(* CODESYS project tc3_hbi_cylinder.library
   Placeholder: Tc3_HBI_Cylinder
   Title: Tc3_HBI_Cylinder
   Version: 3.5.3.6
   DefaultNamespace: Tc3_HBI_Cylinder
   Company: BeckHoff SG

Project tree, tasks and I/O mapping:
  libraries: Tc2_Standard, * (Beckhoff Automation GmbH); Tc2_System, * (Beckhoff Automation GmbH); Tc2_Utilities, * (Beckhoff Automation GmbH); Tc3_HBI_System, * (BeckHoff)
  04_Cylinder/
    DUTs/
      data type _ST_Cylinder
      data type _ST_Cylinder_Status
      data type ST_Cylinder
    ITFs/
      interface I_Cylinder: M_nExtend, M_nOff, M_nRetract, M_nSetOutputOff, P_ipExtend, P_ipRetract, P_nExtendAlarmID, P_nRetractAlarmID, P_opExtend, P_opRetract, P_SensorDelay, P_sExtAlarmDesc, P_sMessage, P_sRetAlarmDesc, P_Timeout
    POUs/
      function block FB_Cylinder [ST]: M_nExtend, M_nOff, M_nReset, M_nRetract, M_nSetOutputOff, P_ipExtend, P_ipRetract, P_nExtendAlarmID, P_nRetractAlarmID, P_opExtend, P_opRetract, P_SensorDelay, P_sExtAlarmDesc, P_sMessage, P_sRetAlarmDesc, P_Timeout
  05_Vacuum/
    DUTs/
      data type _ST_Vacuum
      data type _ST_Vacuum_Status
      data type ST_Vacuum
    ITFs/
      interface I_Vacuum: M_nOff, M_nSetOutputOff, M_nVacuumOff, M_nVacuumOn, P_ipVacuumOff, P_ipVacuumOn, P_nVacOffAlarmID, P_nVacOnAlarmID, P_opVacuumOff, P_opVacuumOn, P_SensorDelay, P_sMessage, P_sVacOffAlarmDesc, P_sVacOnAlarmDesc, P_Timeout
    POUs/
      function block FB_Vacuum [ST]: M_nOff, M_nReset, M_nSetOutputOff, M_nVacuumOff, M_nVacuumOn, P_ipVacuumOff, P_ipVacuumOn, P_nVacOffAlarmID, P_nVacOnAlarmID, P_opVacuumOff, P_opVacuumOn, P_SensorDelay, P_sMessage, P_sVacOffAlarmDesc, P_sVacOnAlarmDesc, P_Timeout
  06_Purge/
    DUTs/
      data type _ST_Purge
      data type _ST_Purge_Status
      data type ST_Purge
    ITFs/
      interface I_Purge: M_nOff, M_nPurgeOff, M_nPurgeOn, M_nSetOutputOff, P_ipPurgeOff, P_ipPurgeOn, P_nPurgeOffAlarmID, P_nPurgeOnAlarmID, P_opPurgeOff, P_opPurgeOn, P_SensorDelay, P_sMessage, P_sPurgeOffAlarmDesc, P_sPurgeOnAlarmDesc, P_Timeout
    POUs/
      function block FB_Purge [ST]: M_nOff, M_nPurgeOff, M_nPurgeOn, M_nReset, M_nSetOutputOff, P_ipPurgeOff, P_ipPurgeOn, P_nPurgeOffAlarmID, P_nPurgeOnAlarmID, P_opPurgeOff, P_opPurgeOn, P_SensorDelay, P_sMessage, P_sPurgeOffAlarmDesc, P_sPurgeOnAlarmDesc, P_Timeout
  07_VacuumPurge/
    DUTs/
      data type _ST_VacuumPurge
      data type _ST_VacuumPurge_Status
      data type ST_VacuumPurge
    ITFs/
      interface I_VacuumPurge: M_nNeutral, M_nPurgeOn, M_nVacuumOn
    POUs/
      function block FB_VacuumPurge [ST]: M_nNeutral, M_nOff, M_nPurgeOff, M_nPurgeOn, M_nSetOutputOff, M_nVacuumOff, M_nVacuumOn, P_ipPurgeOff, P_ipPurgeOn, P_ipVacuumOff, P_ipVacuumOn, P_nPurgeOffAlarmID, P_nPurgeOnAlarmID, P_nVacOffAlarmID, P_nVacOnAlarmID, P_opPurgeOff, P_opPurgeOn, P_opVacuumOff, P_opVacuumOn, P_PurgeTimeout, P_SensorDelay, P_sMessage, P_sPurgeOffAlarmDesc, P_sPurgeOnAlarmDesc, P_sVacOffAlarmDesc, P_sVacOnAlarmDesc, P_Timeout, P_VacuumTimeout
  Version/
    global variables Global_Version
*)

// 04_Cylinder/DUTs/_ST_Cylinder
TYPE _ST_Cylinder EXTENDS ST_Basic :
STRUCT
	;
END_STRUCT
END_TYPE

// 04_Cylinder/DUTs/_ST_Cylinder_Status
TYPE _ST_Cylinder_Status :
STRUCT
	ipExtend	: BOOL;
	ipRetract	: BOOL;
	opExtend	: BOOL;
	opRetract	: BOOL;
	M_nExtend: UDINT;
	M_nRetract: UDINT;
	M_nOff: UDINT;
END_STRUCT
END_TYPE

// 04_Cylinder/DUTs/ST_Cylinder
TYPE ST_Cylinder EXTENDS ST_Basic :
STRUCT
	bExtend		: BOOL;
	bRetract	: BOOL;
	udiExtendAlarmID: UDINT;
	udiRetractAlarmID: UDINT;
	sExtendAlarmDesc: STRING(80);
	sRetractAlarmDesc: STRING(80);
	sMessage: STRING(80);
	Timeout	: TIME:= T#5S;
	SensorDelay: TIME:= T#3S;
	stStatus: _ST_Cylinder_Status;
END_STRUCT
END_TYPE

// 05_Vacuum/DUTs/_ST_Vacuum
TYPE _ST_Vacuum EXTENDS ST_Basic :
STRUCT
	;
END_STRUCT
END_TYPE

// 05_Vacuum/DUTs/_ST_Vacuum_Status
TYPE _ST_Vacuum_Status :
STRUCT
	ipVacuumOn		: BOOL;
	ipVacuumOff		: BOOL;
	opVacuumOn		: BOOL;
	opVacuumOff		: BOOL;
	M_nVacuumOff: UDINT;
	M_nVacuumOn: UDINT;
	M_nOff: UDINT;
END_STRUCT
END_TYPE

// 05_Vacuum/DUTs/ST_Vacuum
TYPE ST_Vacuum EXTENDS ST_Basic :
STRUCT
	bVacuumOn		: BOOL;
	bVacuumOff		: BOOL;
	udiVacOffAlarmID: UDINT;
	udiVacOnAlarmID: UDINT;
	sVacOffAlarmDesc: STRING(80);
	sVacOnAlarmDesc: STRING(80);
	sMessage: STRING(80);
	Timeout	: TIME:= T#5S;
	SensorDelay: TIME:= T#3S;
	stStatus: _ST_Vacuum_Status;
END_STRUCT
END_TYPE

// 06_Purge/DUTs/_ST_Purge
TYPE _ST_Purge EXTENDS ST_Basic :
STRUCT
	;
END_STRUCT
END_TYPE

// 06_Purge/DUTs/_ST_Purge_Status
TYPE _ST_Purge_Status :
STRUCT
	ipPurgeOn		: BOOL;
	ipPurgeOff		: BOOL;
	opPurgeOn		: BOOL;
	opPurgeOff		: BOOL;
	M_nPurgeOff: UDINT;
	M_nPurgeOn: UDINT;
	M_nOff: UDINT;
END_STRUCT
END_TYPE

// 06_Purge/DUTs/ST_Purge
TYPE ST_Purge EXTENDS ST_Basic :
STRUCT
	bPurgeOn		: BOOL;
	bPurgeOff		: BOOL;
	udiPurgeOffAlarmID: UDINT;
	udiPurgeOnAlarmID: UDINT;
	sPurgeOffAlarmDesc: STRING(80);
	sPurgeOnAlarmDesc: STRING(80);
	sMessage: STRING(80);
	Timeout		: TIME:= T#5S;
	SensorDelay	: TIME:= T#3S;	
	stStatus: _ST_Purge_Status;
END_STRUCT
END_TYPE

// 07_VacuumPurge/DUTs/_ST_VacuumPurge
TYPE _ST_VacuumPurge EXTENDS _ST_Purge :
STRUCT
	;
END_STRUCT
END_TYPE

// 07_VacuumPurge/DUTs/_ST_VacuumPurge_Status
TYPE _ST_VacuumPurge_Status :
STRUCT
	;
END_STRUCT
END_TYPE

// 07_VacuumPurge/DUTs/ST_VacuumPurge
TYPE ST_VacuumPurge :
STRUCT
	;
END_STRUCT
END_TYPE

// Version/Global_Version
{attribute 'TcGenerated'}
{attribute 'no-analysis'}
{attribute 'linkalways'}
// This function has been automatically generated from the project information.
VAR_GLOBAL CONSTANT
	{attribute 'const_non_replaced'}
	stLibVersion_Tc3_HBI_Cylinder : ST_LibVersion := (iMajor := 3, iMinor := 5, iBuild := 3, iRevision := 6, sVersion := '3.5.3.6');
END_VAR

// 04_Cylinder/ITFs/I_Cylinder
INTERFACE I_Cylinder EXTENDS Tc3_HBI_System.I_Basic

METHOD M_nExtend : UDINT
VAR_INPUT
	bExecute: BOOL;
END_VAR
END_METHOD

METHOD M_nOff : UDINT
VAR_INPUT
END_VAR
END_METHOD

METHOD M_nRetract : UDINT
VAR_INPUT
	bExecute: BOOL;
END_VAR
END_METHOD

METHOD M_nSetOutputOff : UDINT
VAR_INPUT
END_VAR
END_METHOD

PROPERTY P_ipExtend : BOOL
GET
END_GET
SET
END_SET
END_PROPERTY

PROPERTY P_ipRetract : BOOL
GET
END_GET
SET
END_SET
END_PROPERTY

PROPERTY P_nExtendAlarmID : UDINT
SET
END_SET
END_PROPERTY

PROPERTY P_nRetractAlarmID : UDINT
SET
END_SET
END_PROPERTY

PROPERTY P_opExtend : BOOL
GET
END_GET
SET
END_SET
END_PROPERTY

PROPERTY P_opRetract : BOOL
GET
END_GET
SET
END_SET
END_PROPERTY

PROPERTY P_SensorDelay : TIME
SET
END_SET
END_PROPERTY

PROPERTY P_sExtAlarmDesc : STRING
SET
END_SET
END_PROPERTY

PROPERTY P_sMessage : STRING
GET
END_GET
END_PROPERTY

PROPERTY P_sRetAlarmDesc : STRING
SET
END_SET
END_PROPERTY

PROPERTY P_Timeout : TIME
SET
END_SET
END_PROPERTY

END_INTERFACE

// 04_Cylinder/POUs/FB_Cylinder
//------------------------------------------------------------------------------------------
//                                                                                        	
//***************************** Beckhoff TwinCAT Examples **********************************
//                                                                                        	
//************************************* WARNING ********************************************
// This program is only an example. If it is used as a control program in any real        	
// application, Beckhoff is not responsible for any malfunction, loss or damage           	
// which could arise by using this program!                                               	
//                                                                                        	
//*************************************  Program Info. *************************************
//                                                                                        	
// PLC program name:       	FB_Cylinder (FB)                                          	
// Hardware platform:      	TwinCat PTP v3.1.4022				                          	                                  	
//                                                                                        	
// ======================================================================================== 
//         Version       Date                        Remarks                              	
// ======================================================================================== 
//         3.1.1.1      01 March 2018                First release of this example  
//         3.1.1.2      05 March 2018                Next release of this example  
//         3.2.1.1      09 March 2018                Next release of this example  
//         3.2.2.0      09 April 2018                Next release of this example 
//         3.2.2.1      13 April 2018                Next release of this example    
// ======================================================================================== 
//                                                                                        	
//******************************* Aims OF this PLC PROGRAM *********************************
//                                                                                        	
// 	3.2.2.0 added message for cylinder alarm					 			                                      	
//	3.2.2.1 sloved the cylinder timer start when alarm reset always trigger															                      	
//  3.3.3.1 add property for get set to send status out  
//	3.5.1.1 user config alarm decription & ID  
//	3.5.3.2 sensor delay set to 0    
//	3.5.3.4 if switch extend and retract, init extend or retract                                                                              	
//----------------------------------------------------------------------------------------- 
FUNCTION_BLOCK FB_Cylinder EXTENDS FB_Basic IMPLEMENTS I_Cylinder
VAR	
	FB_Cylinder_M_nExetend_iState	: INT;
	FB_Cylinder_M_nExetend_bExecute	: BOOL;
	FB_Cylinder_M_nExetend_fbExecute_R_TRIG: Tc2_Standard.R_TRIG;
	
	FB_Cylinder_M_nRetract_iState	: INT;
	FB_Cylinder_M_nRetract_bExecute	: BOOL;
	FB_Cylinder_M_nRetract_fbExecute_R_TRIG: Tc2_Standard.R_TRIG;
	
	FB_Cylinder_M_nReset_iState	: INT;
	FB_Cylinder_M_nReset_bExecute	: BOOL;
	FB_Cylinder_M_nReset_fbExecute_R_TRIG: Tc2_Standard.R_TRIG;
	FB_Cylinder_M_nReset_nStatus	: UDINT;
	
	FB_Cylinder_ipExtend	: BOOL;
	FB_Cylinder_ipRetract	: BOOL;
	FB_Cylinder_opExtend	: BOOL;
	FB_Cylinder_opRetract	: BOOL;
	FB_Cylinder_Timeout		: TIME:= T#5S;
	FB_Cylinder_SensorDelay	: TIME:= T#0MS;
	FB_Cylinder_sMessage		: STRING(80);
	FB_Cylinder_sExtAlarmDesc	: STRING(80):='Extend Error';
	FB_Cylinder_sRetAlarmDesc	: STRING(80):= 'Retract Error';
	FB_Cylinder_nExtAlarmID		: UDINT:= 999;
	FB_Cylinder_nRetAlarmID		: UDINT:= 999;
	
	FB_Cylinder_fbTimeout: Tc2_Standard.TON;
	FB_Cylinder_fbSensorDelay: Tc2_Standard.TON;
END_VAR

// =========================================================
	

// =========================================================

METHOD M_nExtend : UDINT
VAR_INPUT	
	bExecute		: BOOL;
END_VAR
// =========================================================
	// Local variables
FB_Cylinder_M_nExetend_bExecute:= bExecute;		

// =========================================================		
	// Reset
	IF _bReset THEN
		IF _bError THEN;
			FB_Cylinder_sMessage:= '';
			IF FB_Cylinder_M_nExetend_bExecute THEN
				FB_Cylinder_M_nExetend_iState:= 01;
				ELSE FB_Cylinder_M_nExetend_iState:= 00;
			END_IF
		END_IF	
	END_IF

// =========================================================
	// Extend request
	FB_Cylinder_M_nExetend_fbExecute_R_TRIG(CLK:= FB_Cylinder_M_nExetend_bExecute, Q=> );
	
	IF FB_Cylinder_M_nExetend_fbExecute_R_TRIG.Q THEN
		M_nRetract(bExecute:= FALSE);
		FB_Cylinder_M_nExetend_iState:= 01;
	END_IF
	
// =========================================================
	// Both extend and retract are triggered
	IF FB_Cylinder_M_nRetract_bExecute AND FB_Cylinder_M_nExetend_bExecute THEN
		FB_Cylinder_M_nExetend_iState:= 9999;
	END_IF
		
// =========================================================
	// State machine
		
CASE FB_Cylinder_M_nExetend_iState OF 
	
	00: // Do nothing
		M_nExtend:= Tc3_HBI_System.cIDLE;
		
	01:// Reset timer
		M_nExtend:= Tc3_HBI_System.cRUNNING;
		
		FB_Cylinder_fbTimeout(IN:= FALSE, PT:= FB_Cylinder_Timeout, Q=> , ET=> );
		FB_Cylinder_fbSensorDelay(IN:= FALSE, PT:= FB_Cylinder_SensorDelay, Q=> , ET=> );
		
		IF FB_Cylinder_M_nExetend_bExecute THEN
			FB_Cylinder_M_nExetend_iState:= FB_Cylinder_M_nExetend_iState+1;
		ELSE 
			FB_Cylinder_M_nExetend_iState:= 0;
		END_IF
		
	02:// Starting
		M_nExtend:= Tc3_HBI_System.cSTARTING;
		
		IF _bReset THEN
			FB_Cylinder_M_nExetend_iState:= FB_Cylinder_M_nExetend_iState-1;
			ELSIF FB_Cylinder_M_nExetend_bExecute THEN
				FB_Cylinder_M_nExetend_iState:= FB_Cylinder_M_nExetend_iState+1;				
					ELSE FB_Cylinder_M_nExetend_iState:= 00;
		END_IF
	
	03: // Extend 
		M_nExtend:= Tc3_HBI_System.cRUNNING;
		
		FB_Cylinder_opRetract:= FALSE;
		FB_Cylinder_opExtend:= TRUE;	
		FB_Cylinder_fbTimeout(IN:= TRUE, PT:= FB_Cylinder_Timeout, Q=> , ET=> );
		FB_Cylinder_fbSensorDelay(IN:= FB_Cylinder_ipExtend, PT:= FB_Cylinder_SensorDelay, Q=> , ET=> );
		
		IF FB_Cylinder_fbSensorDelay.Q THEN
			FB_Cylinder_M_nExetend_iState:= FB_Cylinder_M_nExetend_iState+1;
			ELSIF FB_Cylinder_fbTimeout.Q THEN
//					M_nError(nErrorID:= FB_Cylinder_nExtAlarmID);
//					FB_Cylinder_sMessage:= CONCAT(CONCAT(UDINT_TO_STRING(FB_Cylinder_nExtAlarmID),'>'),
//														CONCAT('>',FB_Cylinder_sExtAlarmDesc));
					FB_Cylinder_M_nExetend_iState:= 999;
				ELSIF NOT FB_Cylinder_M_nExetend_bExecute THEN
					FB_Cylinder_fbTimeout(IN:= FALSE, PT:= FB_Cylinder_Timeout, Q=> , ET=> );
					FB_Cylinder_fbSensorDelay(IN:= FALSE, PT:= FB_Cylinder_SensorDelay, Q=> , ET=> );
//					FB_Cylinder_opExtend:= FALSE;
					FB_Cylinder_M_nExetend_iState:= 0;
		END_IF
	
	04: // Extend done
		M_nExtend:= Tc3_HBI_System.cCOMPLETE;
		
		IF NOT FB_Cylinder_M_nExetend_bExecute THEN
			FB_Cylinder_M_nExetend_iState:= 00;
		END_IF		
		
	999: // Error state
		M_nExtend:= Tc3_HBI_System.cABORTED;
		
		M_nError(nErrorID:= FB_Cylinder_nExtAlarmID);
		FB_Cylinder_sMessage:= CONCAT(CONCAT(UDINT_TO_STRING(FB_Cylinder_nExtAlarmID),'>'),
											CONCAT('>',FB_Cylinder_sExtAlarmDesc));
		
		FB_Cylinder_fbSensorDelay(IN:= FALSE, PT:= T#0S, Q=> , ET=> );
		FB_Cylinder_fbTimeout(IN:= FALSE, PT:= T#0S, Q=> , ET=> );
		
		IF NOT FB_Cylinder_M_nExetend_bExecute THEN
			FB_Cylinder_M_nExetend_iState:= 0;
		END_IF
		
	9999: // Parameter error state
		M_nExtend:= Tc3_HBI_System.cPARAMETER_ERROR;
		M_nError(nErrorID:= Tc3_HBI_System.cPARAMETER_ERROR);
		FB_Cylinder_sMessage:= 'Both extend and retract are triggered';
	
	ELSE
		FB_Cylinder_M_nExetend_iState:= 0;
		
END_CASE
// =========================================================
END_METHOD

METHOD M_nOff : UDINT
VAR_INPUT
END_VAR
// =========================================================
	M_nExtend(bExecute:= FALSE);
	M_nRetract(bExecute:= FALSE);
	
	M_nOff:= Tc3_HBI_System.cCOMPLETE;
// =========================================================
END_METHOD

//	The result of the method is an unsigned double integer
//	0 = idle 
//	1 = coupled
//	2 = starting
//	3 = running
//	4 = aborted
// 	5 = no hardware connected
//  6 = Spare
//	7 = pointer or index error
//	8 = mapping error
//	9 = parameter error
//	10 = complete
//	Any other number = ErrorID
METHOD PUBLIC M_nReset : UDINT
VAR_INPUT
	bExecute: BOOL;
END_VAR
// =========================================================
	// Local variables
FB_Cylinder_M_nReset_bExecute:= bExecute;

// =========================================================	
	// Fire
FB_Cylinder_M_nReset_fbExecute_R_TRIG(CLK:= FB_Cylinder_M_nReset_bExecute, Q=> );
IF FB_Cylinder_M_nReset_fbExecute_R_TRIG.Q THEN
	SUPER^.M_nReset(bExecute:= FALSE);
	FB_Cylinder_M_nReset_iState:= 01;
END_IF

// =========================================================
	// State machine
	
CASE FB_Cylinder_M_nReset_iState OF
	00: // Init
		;
	01:// Starting
		M_nReset:= Tc3_HBI_System.cSTARTING;
		
		FB_Cylinder_sMessage:= '';
		
		FB_Cylinder_M_nExetend_bExecute:= FALSE;
		FB_Cylinder_M_nExetend_fbExecute_R_TRIG(CLK:= FALSE, Q=> );
		FB_Cylinder_M_nExetend_iState:= 0;
		
		FB_Cylinder_M_nRetract_bExecute:= FALSE;
		FB_Cylinder_M_nRetract_fbExecute_R_TRIG(CLK:= FALSE, Q=> );
		FB_Cylinder_M_nRetract_iState:= 0;
		
		FB_Cylinder_M_nReset_iState:= FB_Cylinder_M_nReset_iState+1;
		
	02:// Running
		M_nReset:= Tc3_HBI_System.cRUNNING;
		FB_Cylinder_M_nReset_nStatus:= SUPER^.M_nReset(bExecute:= TRUE);
		
		// Error 
			IF FB_Cylinder_M_nReset_nStatus > Tc3_HBI_System.cCOMPLETE THEN
				SUPER^.M_nReset(bExecute:= FALSE);		
				FB_Cylinder_M_nReset_iState:= FB_Cylinder_M_nReset_iState+1;
			END_IF

			// Done
			IF FB_Cylinder_M_nReset_nStatus = Tc3_HBI_System.cCOMPLETE THEN
				SUPER^.M_nReset(bExecute:= FALSE);		
				FB_Cylinder_M_nReset_iState:= FB_Cylinder_M_nReset_iState+1;
			END_IF
			
	03: // Done
		M_nReset:= Tc3_HBI_System.cCOMPLETE;
		
			IF NOT FB_Cylinder_M_nReset_bExecute THEN
				SUPER^.M_nReset(bExecute:= FALSE);		
				FB_Cylinder_M_nReset_iState:= 000;
			END_IF
	ELSE 
		FB_Cylinder_M_nReset_iState:= 0;
END_CASE
END_METHOD

METHOD M_nRetract : UDINT
VAR_INPUT	
	bExecute	: BOOL;
END_VAR
// =========================================================
	// Local variables		
FB_Cylinder_M_nRetract_bExecute:= bExecute;

// =========================================================		
	// Reset
	IF _bReset THEN
		IF _bError THEN;
			FB_Cylinder_sMessage:= '';
			IF FB_Cylinder_M_nRetract_bExecute THEN
				FB_Cylinder_M_nRetract_iState:= 01;
				ELSE FB_Cylinder_M_nRetract_iState:= 00;
			END_IF
		END_IF	
	END_IF

// =========================================================
	// Retract request
	FB_Cylinder_M_nRetract_fbExecute_R_TRIG(CLK:= FB_Cylinder_M_nRetract_bExecute, Q=> );
	
	IF FB_Cylinder_M_nRetract_fbExecute_R_TRIG.Q THEN
		M_nExtend(bExecute:= FALSE);
		FB_Cylinder_M_nRetract_iState:= 01;
	END_IF
	
// =========================================================
	// Both extend and retract are triggered
	IF FB_Cylinder_M_nRetract_bExecute AND FB_Cylinder_M_nExetend_bExecute THEN
		FB_Cylinder_M_nRetract_iState:= 9999;
	END_IF
		
// =========================================================
	// State machine
		
CASE FB_Cylinder_M_nRetract_iState OF 
	
	00: // Do nothing
		M_nRetract:= Tc3_HBI_System.cIDLE;
		
	01:// Reset timer
		M_nRetract:= Tc3_HBI_System.cRUNNING;
		
		FB_Cylinder_fbTimeout(IN:= FALSE, PT:= FB_Cylinder_Timeout, Q=> , ET=> );
		FB_Cylinder_fbSensorDelay(IN:= FALSE, PT:= FB_Cylinder_SensorDelay, Q=> , ET=> );
		
		IF FB_Cylinder_M_nRetract_bExecute THEN
			FB_Cylinder_M_nRetract_iState:= FB_Cylinder_M_nRetract_iState+1;
		ELSE 
			FB_Cylinder_M_nRetract_iState:= 0;
		END_IF
		
	02:// Starting
		M_nRetract:= Tc3_HBI_System.cSTARTING;
		
		IF _bReset THEN
			FB_Cylinder_M_nRetract_iState:= FB_Cylinder_M_nRetract_iState-1;
			ELSIF FB_Cylinder_M_nRetract_bExecute THEN
				FB_Cylinder_M_nRetract_iState:= FB_Cylinder_M_nRetract_iState+1;					
					ELSE FB_Cylinder_M_nRetract_iState:= 00;
		END_IF
		
	03: // Retract
		M_nRetract:= Tc3_HBI_System.cRUNNING;
		
		FB_Cylinder_opExtend:= FALSE;
		FB_Cylinder_opRetract:= TRUE;
		FB_Cylinder_fbTimeout(IN:= TRUE, PT:= FB_Cylinder_Timeout, Q=> , ET=> );
		FB_Cylinder_fbSensorDelay(IN:= FB_Cylinder_ipRetract, PT:= FB_Cylinder_SensorDelay, Q=> , ET=> );
		
		IF FB_Cylinder_fbSensorDelay.Q THEN
			FB_Cylinder_M_nRetract_iState:= FB_Cylinder_M_nRetract_iState+1;
			ELSIF FB_Cylinder_fbTimeout.Q THEN
//					M_nError(nErrorID:= FB_Cylinder_nRetAlarmID);
//					FB_Cylinder_sMessage:= CONCAT(CONCAT(UDINT_TO_STRING(FB_Cylinder_nRetAlarmID),'>'),
//														CONCAT('>',FB_Cylinder_sRetAlarmDesc));
					FB_Cylinder_M_nRetract_iState:= 999;
				ELSIF NOT FB_Cylinder_M_nRetract_bExecute THEN
					FB_Cylinder_fbSensorDelay(IN:= FALSE, PT:= T#0S, Q=> , ET=> );
					FB_Cylinder_fbTimeout(IN:= FALSE, PT:= T#0S, Q=> , ET=> );
//					FB_Cylinder_opRetract:= FALSE;
					FB_Cylinder_M_nRetract_iState:= 0;
		END_IF
		
	04: // Retract done
		M_nRetract:= Tc3_HBI_System.cCOMPLETE;
		
		IF NOT FB_Cylinder_M_nRetract_bExecute THEN
			FB_Cylinder_M_nRetract_iState:= 0;
		END_IF
		
	999: // Error state
		M_nRetract:= Tc3_HBI_System.cABORTED;
		
		M_nError(nErrorID:= FB_Cylinder_nRetAlarmID);
		FB_Cylinder_sMessage:= CONCAT(CONCAT(UDINT_TO_STRING(FB_Cylinder_nRetAlarmID),'>'),
											CONCAT('>',FB_Cylinder_sRetAlarmDesc));
		
		FB_Cylinder_fbSensorDelay(IN:= FALSE, PT:= T#0S, Q=> , ET=> );
		FB_Cylinder_fbTimeout(IN:= FALSE, PT:= T#0S, Q=> , ET=> );
		
		IF NOT FB_Cylinder_M_nRetract_bExecute THEN
			FB_Cylinder_M_nRetract_iState:= 0;
		END_IF
		
	9999: // Parameter error state
		M_nRetract:= Tc3_HBI_System.cPARAMETER_ERROR;
		M_nError(nErrorID:= Tc3_HBI_System.cPARAMETER_ERROR);
		FB_Cylinder_sMessage:= 'Both extend and retract are triggered';

	ELSE
		FB_Cylinder_M_nRetract_iState:= 0;
		
END_CASE
// =========================================================
END_METHOD

METHOD M_nSetOutputOff : UDINT
VAR_INPUT
END_VAR
END_METHOD

{warning 'add property implementation'}
PROPERTY P_ipExtend : BOOL
GET
P_ipExtend:= FB_Cylinder_ipExtend;
END_GET
SET
FB_Cylinder_ipExtend := P_ipExtend;
END_SET
END_PROPERTY

{warning 'add property implementation'}
PROPERTY P_ipRetract : BOOL
GET
P_ipRetract:= FB_Cylinder_ipRetract;
END_GET
SET
FB_Cylinder_ipRetract := P_ipRetract;
END_SET
END_PROPERTY

PROPERTY P_nExtendAlarmID : UDINT
SET
FB_Cylinder_nExtAlarmID:= P_nExtendAlarmID;
END_SET
END_PROPERTY

PROPERTY P_nRetractAlarmID : UDINT
SET
FB_Cylinder_nRetAlarmID:= P_nRetractAlarmID;
END_SET
END_PROPERTY

{warning 'add property implementation'}
PROPERTY P_opExtend : BOOL
GET
P_opExtend := FB_Cylinder_opExtend;
END_GET
SET
FB_Cylinder_opExtend:= P_opExtend;
END_SET
END_PROPERTY

{warning 'add property implementation'}
PROPERTY P_opRetract : BOOL
GET
P_opRetract := FB_Cylinder_opRetract;
END_GET
SET
FB_Cylinder_opRetract:= P_opRetract;
END_SET
END_PROPERTY

PROPERTY P_SensorDelay : TIME
SET
FB_Cylinder_SensorDelay:= P_SensorDelay;
END_SET
END_PROPERTY

PROPERTY P_sExtAlarmDesc : STRING
SET
FB_Cylinder_sExtAlarmDesc:= P_sExtAlarmDesc;
END_SET
END_PROPERTY

PROPERTY PUBLIC P_sMessage : string
GET
P_sMessage:= FB_Cylinder_sMessage;
END_GET
END_PROPERTY

PROPERTY P_sRetAlarmDesc : STRING
SET
FB_Cylinder_sRetAlarmDesc:= P_sRetAlarmDesc;
END_SET
END_PROPERTY

{warning 'add property implementation'}
PROPERTY P_Timeout : TIME
SET
FB_Cylinder_Timeout:= P_Timeout;
END_SET
END_PROPERTY

END_FUNCTION_BLOCK

// 05_Vacuum/ITFs/I_Vacuum
INTERFACE I_Vacuum EXTENDS Tc3_HBI_System.I_Basic

METHOD M_nOff : UDINT
VAR_INPUT
END_VAR
END_METHOD

METHOD M_nSetOutputOff : UDINT
VAR_INPUT
END_VAR
END_METHOD

METHOD M_nVacuumOff : UDINT
VAR_INPUT
	bExecute: BOOL;
END_VAR
END_METHOD

METHOD M_nVacuumOn : UDINT
VAR_INPUT
	bExecute: BOOL;
END_VAR
END_METHOD

PROPERTY P_ipVacuumOff : BOOL
GET
END_GET
SET
END_SET
END_PROPERTY

PROPERTY P_ipVacuumOn : BOOL
GET
END_GET
SET
END_SET
END_PROPERTY

PROPERTY P_nVacOffAlarmID : UDINT
SET
END_SET
END_PROPERTY

PROPERTY P_nVacOnAlarmID : UDINT
SET
END_SET
END_PROPERTY

PROPERTY P_opVacuumOff : BOOL
GET
END_GET
SET
END_SET
END_PROPERTY

PROPERTY P_opVacuumOn : BOOL
GET
END_GET
SET
END_SET
END_PROPERTY

PROPERTY P_SensorDelay : TIME
SET
END_SET
END_PROPERTY

PROPERTY P_sMessage : STRING
GET
END_GET
END_PROPERTY

PROPERTY P_sVacOffAlarmDesc : string
SET
END_SET
END_PROPERTY

PROPERTY P_sVacOnAlarmDesc : STRING
SET
END_SET
END_PROPERTY

PROPERTY P_Timeout : TIME
SET
END_SET
END_PROPERTY

END_INTERFACE

// 05_Vacuum/POUs/FB_Vacuum
//------------------------------------------------------------------------------------------
//                                                                                        	
//***************************** Beckhoff TwinCAT Examples **********************************
//                                                                                        	
//************************************* WARNING ********************************************
// This program is only an example. If it is used as a control program in any real        	
// application, Beckhoff is not responsible for any malfunction, loss or damage           	
// which could arise by using this program!                                               	
//                                                                                        	
//*************************************  Program Info. *************************************
//                                                                                        	
// PLC program name:       	FB_Vacuum (FB)                                          	
// Hardware platform:      	TwinCat PTP v3.1.4022				                          	                                  	
//                                                                                        	
// ======================================================================================== 
//         Version       Date                        Remarks                              	
// ======================================================================================== 
//         3.1.1.1      01 March 2018                First release of this example 
//         3.1.1.2      05 March 2018                Next release of this example    
//         3.2.1.1      09 March 2018                Next release of this example 
//         3.3.1.1      09 March 2018                Next release of this example  
// ======================================================================================== 
//                                                                                        	
//******************************* Aims OF this PLC PROGRAM *********************************
//                                                                                        	
// 	3.2.2.0 added message for vacuum alarm 						 			                                      	
//	3.5.3.1 Off output once error																                      	
//                                                                                        	
//----------------------------------------------------------------------------------------- 
FUNCTION_BLOCK FB_Vacuum EXTENDS FB_Basic IMPLEMENTS I_Vacuum
VAR 
	FB_Vacuum_M_nVacuumOff_iState	: INT;
	FB_Vacuum_M_nVacuumOff_bExecute	: BOOL;
	FB_Vacuum_M_nVacuumOff_fbExecute_R_TRIG: Tc2_Standard.R_TRIG;
	
	FB_Vacuum_M_nVacuumOn_iState	: INT;
	FB_Vacuum_M_nVacuumOn_bExecute	: BOOL;
	FB_Vacuum_M_nvacuumOn_fbExecute_R_TRIG: Tc2_Standard.R_TRIG;
	
	FB_Vacuum_M_nReset_iState	: INT;
	FB_Vacuum_M_nReset_bExecute	: BOOL;
	FB_Vacuum_M_nReset_fbExecute_R_TRIG: Tc2_Standard.R_TRIG;
	FB_Vacuum_M_nReset_nStatus	: UDINT;
	
	FB_Vacuum_ipVacuumOn	: BOOL;
	FB_Vacuum_ipVacuumOff	: BOOL;
	FB_Vacuum_opVacuumOn	: BOOL;
	FB_Vacuum_opVacuumOff	: BOOL;
	
	FB_Vacuum_Timeout		: TIME:= T#5S;
	FB_Vacuum_SensorDelay	: TIME:= T#0MS;
	FB_Vacuum_sMessage		: STRING(80);
	
	FB_Vacuum_sVacOffAlarmDesc	: STRING(80):='Vacuum Off Error';
	FB_Vacuum_sVacOnAlarmDesc	: STRING(80):= 'Vacuum On Error';
	FB_Vacuum_nVacOffAlarmID	: UDINT:= 999;
	FB_Vacuum_nVacOnAlarmID		: UDINT:= 999;
	
	FB_Vacuum_fbTimeout: Tc2_Standard.TON;
	FB_Vacuum_fbSensorDelay: Tc2_Standard.TON;	
END_VAR

{warning 'add method implementation'}
METHOD M_nOff : UDINT
// =========================================================
M_nVacuumOff(bExecute:= FALSE);
M_nVacuumOn(bExecute:= FALSE);

M_nOff:= Tc3_HBI_System.cCOMPLETE;
// =========================================================
END_METHOD

//	The result of the method is an unsigned double integer
//	0 = idle 
//	1 = coupled
//	2 = starting
//	3 = running
//	4 = aborted
// 	5 = no hardware connected
//  6 = Spare
//	7 = pointer or index error
//	8 = mapping error
//	9 = parameter error
//	10 = complete
//	Any other number = ErrorID
METHOD PUBLIC M_nReset : UDINT
VAR_INPUT
	bExecute: BOOL;
END_VAR
// =========================================================
	// Local variables
FB_Vacuum_M_nReset_bExecute:= bExecute;

// =========================================================	
	// Fire
FB_Vacuum_M_nReset_fbExecute_R_TRIG(CLK:= FB_Vacuum_M_nReset_bExecute, Q=> );
IF FB_Vacuum_M_nReset_fbExecute_R_TRIG.Q THEN
	SUPER^.M_nReset(bExecute:= FALSE);
	FB_Vacuum_M_nReset_iState:= 01;
END_IF

// =========================================================
	// State machine
	
CASE FB_Vacuum_M_nReset_iState OF
	00: // Init
		;
		
	01:// Starting
		M_nReset:= Tc3_HBI_System.cSTARTING;
		
		FB_Vacuum_sMessage:= '';
		
		FB_Vacuum_M_nVacuumOff_bExecute:= FALSE;
		FB_Vacuum_M_nVacuumOff_fbExecute_R_TRIG(CLK:= FALSE, Q=> );
		FB_Vacuum_M_nVacuumOff_iState:= 0;
		
		FB_Vacuum_M_nVacuumOn_bExecute:= FALSE;
		FB_Vacuum_M_nVacuumOn_fbExecute_R_TRIG(CLK:= FALSE, Q=> );
		FB_Vacuum_M_nVacuumOn_iState:= 0;
		
		FB_Vacuum_M_nReset_iState:= FB_Vacuum_M_nReset_iState+1;
		
	02:// Running
		M_nReset:= Tc3_HBI_System.cRUNNING;
		
		FB_Vacuum_M_nReset_nStatus:= SUPER^.M_nReset(bExecute:= TRUE);
		
		// Error 
			IF FB_Vacuum_M_nReset_nStatus > Tc3_HBI_System.cCOMPLETE THEN
				SUPER^.M_nReset(bExecute:= FALSE);		
				FB_Vacuum_M_nReset_iState:= FB_Vacuum_M_nReset_iState+1;
			END_IF

		// Done
			IF FB_Vacuum_M_nReset_nStatus = Tc3_HBI_System.cCOMPLETE THEN
				SUPER^.M_nReset(bExecute:= FALSE);		
				FB_Vacuum_M_nReset_iState:= FB_Vacuum_M_nReset_iState+1;
			END_IF
			
	03: // Done
		M_nReset:= Tc3_HBI_System.cCOMPLETE;
			IF NOT FB_Vacuum_M_nReset_bExecute THEN
				SUPER^.M_nReset(bExecute:= FALSE);		
				FB_Vacuum_M_nReset_iState:= 000;
			END_IF
	ELSE 
		FB_Vacuum_M_nReset_iState:= 0;
END_CASE
END_METHOD

METHOD M_nSetOutputOff : UDINT
VAR_INPUT
END_VAR
END_METHOD

{warning 'add method implementation'}
METHOD M_nVacuumOff : UDINT
VAR_INPUT
	bExecute	: BOOL;
END_VAR
// =========================================================
		// Local variables
FB_Vacuum_M_nVacuumOff_bExecute:= bExecute;		

// =========================================================		
		// Reset
IF _bReset THEN
	IF _bError THEN;
		FB_Vacuum_sMessage:= '';
		IF FB_Vacuum_M_nVacuumOff_bExecute THEN
			FB_Vacuum_M_nVacuumOff_iState:= 01;
			ELSE FB_Vacuum_M_nVacuumOff_iState:= 00;
		END_IF
	END_IF	
END_IF

// =========================================================
		// Vacuum off requested
	FB_Vacuum_M_nVacuumOff_fbExecute_R_TRIG(CLK:= FB_Vacuum_M_nVacuumOff_bExecute, Q=> );
	
	IF FB_Vacuum_M_nVacuumOff_fbExecute_R_TRIG.Q THEN
		M_nVacuumOn(bExecute:= FALSE);
		FB_Vacuum_M_nVacuumOff_iState:= 01;
	END_IF
	
// =========================================================
	// Both vacuum on and vacuum off are triggered
	IF FB_Vacuum_M_nVacuumOff_bExecute AND FB_Vacuum_M_nVacuumOn_bExecute THEN
		FB_Vacuum_M_nVacuumOff_iState:= 9999;
	END_IF
		
// =========================================================
		// Vacuum off state
		
CASE FB_Vacuum_M_nVacuumOff_iState OF 
	
	00: // Do nothing
		M_nVacuumOff:= Tc3_HBI_System.cIDLE;
		
	01:// Reset timer
		M_nVacuumOff:= Tc3_HBI_System.cRUNNING;
		FB_Vacuum_fbTimeout(IN:= FALSE, PT:= FB_Vacuum_Timeout, Q=> , ET=> );
		FB_Vacuum_fbSensorDelay(IN:= FALSE, PT:= FB_Vacuum_SensorDelay, Q=> , ET=> );
		
		FB_Vacuum_M_nVacuumOff_iState:= FB_Vacuum_M_nVacuumOff_iState+1;
		
	02:// Starting
		M_nVacuumOff:= Tc3_HBI_System.cSTARTING;
		
		IF _bReset THEN
			FB_Vacuum_M_nVacuumOff_iState:= FB_Vacuum_M_nVacuumOff_iState-1;
			ELSIF FB_Vacuum_M_nVacuumOff_bExecute THEN
				FB_Vacuum_M_nVacuumOff_iState:= FB_Vacuum_M_nVacuumOff_iState+1;
				ELSE FB_Vacuum_M_nVacuumOff_iState:= 00;
		END_IF
		
	03: // Vacuum off
		M_nVacuumOff:= Tc3_HBI_System.cRUNNING;
		
		FB_Vacuum_opVacuumOn:= FALSE;
		FB_Vacuum_opVacuumOff:= TRUE;
		FB_Vacuum_fbTimeout(IN:= TRUE, PT:= FB_Vacuum_Timeout, Q=> , ET=> );
		FB_Vacuum_fbSensorDelay(IN:= FB_Vacuum_ipVacuumOff, PT:= FB_Vacuum_SensorDelay, Q=> , ET=> );
		
		IF FB_Vacuum_fbSensorDelay.Q THEN
			FB_Vacuum_M_nVacuumOff_iState:= FB_Vacuum_M_nVacuumOff_iState+1;
			ELSE 
				IF FB_Vacuum_fbTimeout.Q THEN
//					M_nError(nErrorID:= FB_Vacuum_nVacOffAlarmID);
//					FB_Vacuum_sMessage:= CONCAT(CONCAT(UDINT_TO_STRING(FB_Vacuum_nVacOffAlarmID),'>'),
//														CONCAT('>',FB_Vacuum_svacOffAlarmDesc));
					FB_Vacuum_M_nVacuumOff_iState:= 999;
				END_IF
		END_IF
		
	04: // Vacuum done
		M_nVacuumOff:= Tc3_HBI_System.cCOMPLETE;
		
		IF NOT FB_Vacuum_M_nVacuumOff_bExecute THEN
			FB_Vacuum_M_nVacuumOff_iState:= 0;
		END_IF
		
	999: // Error state
		M_nVacuumOff:= Tc3_HBI_System.cABORTED;
		
		FB_Vacuum_opVacuumOn:= FALSE;
		FB_Vacuum_opVacuumOff:= FALSE;
		
		M_nError(nErrorID:= FB_Vacuum_nVacOffAlarmID);
		FB_Vacuum_sMessage:= CONCAT(CONCAT(UDINT_TO_STRING(FB_Vacuum_nVacOffAlarmID),'>'),
											CONCAT('>',FB_Vacuum_svacOffAlarmDesc));
		
		FB_Vacuum_fbTimeout(IN:= FALSE, PT:= T#0S, Q=> , ET=> );
		FB_Vacuum_fbSensorDelay(IN:= FALSE, PT:= T#0S, Q=> , ET=> );
		
		IF NOT FB_Vacuum_M_nVacuumOff_bExecute THEN
			FB_Vacuum_M_nVacuumOff_iState:= 0;
		END_IF
		
	9999: // Parameter error state
		M_nVacuumOff:= Tc3_HBI_System.cPARAMETER_ERROR;
		M_nError(nErrorID:= Tc3_HBI_System.cPARAMETER_ERROR);
		FB_Vacuum_sMessage:= 'Both vacuum on and vacuum off are triggered';
	
ELSE
	FB_Vacuum_M_nVacuumOff_iState:= 00;
	
END_CASE
// =========================================================
END_METHOD

{warning 'add method implementation'}
METHOD M_nVacuumOn : UDINT
VAR_INPUT
	bExecute	: BOOL;
END_VAR
// =========================================================
		// Local variables
FB_Vacuum_M_nVacuumOn_bExecute:= bExecute;		

// =========================================================		
		// Reset
IF _bReset THEN
	IF _bError THEN;
		FB_Vacuum_sMessage:= '';
		IF FB_Vacuum_M_nVacuumOn_bExecute THEN
			FB_Vacuum_M_nVacuumOn_iState:= 01;
			ELSE FB_Vacuum_M_nVacuumOn_iState:= 00;
		END_IF
	END_IF	
END_IF

// =========================================================
		// Vacuum on requested
	FB_Vacuum_M_nVacuumOn_fbExecute_R_TRIG(CLK:= FB_Vacuum_M_nVacuumOn_bExecute, Q=> );
	
	IF FB_Vacuum_M_nVacuumOn_fbExecute_R_TRIG.Q THEN
		M_nVacuumOff(bExecute:= FALSE);
		FB_Vacuum_M_nVacuumOn_iState:= 01;
	END_IF

// =========================================================
	// Both vacuum on and vacuum off are triggered
	IF FB_Vacuum_M_nVacuumOff_bExecute AND FB_Vacuum_M_nVacuumOn_bExecute THEN
		FB_Vacuum_M_nVacuumOn_iState:= 9999;
	END_IF
		
// =========================================================
		// Vacuum on state
		
CASE FB_Vacuum_M_nVacuumOn_iState OF 
	
	00: // Do nothing
		M_nVacuumOn:= Tc3_HBI_System.cIDLE;
		
	01:// Reset timer
		M_nVacuumOn:= Tc3_HBI_System.cRUNNING;
		
		FB_Vacuum_fbTimeout(IN:= FALSE, PT:= FB_Vacuum_Timeout, Q=> , ET=> );
		FB_Vacuum_fbSensorDelay(IN:= FALSE, PT:= FB_Vacuum_SensorDelay, Q=> , ET=> );
		
		FB_Vacuum_M_nVacuumOn_iState:= FB_Vacuum_M_nVacuumOn_iState+1;
		
	02:// Starting
		M_nVacuumOn:= Tc3_HBI_System.cSTARTING;
		
		IF _bReset THEN
			FB_Vacuum_M_nVacuumOn_iState:= FB_Vacuum_M_nVacuumOn_iState-1;
			ELSIF FB_Vacuum_M_nVacuumOn_bExecute THEN
				FB_Vacuum_M_nVacuumOn_iState:= FB_Vacuum_M_nVacuumOn_iState+1;
				ELSE FB_Vacuum_M_nVacuumOn_iState:= 00;
		END_IF
		
	03: // Vacuum on
		M_nVacuumOn:= Tc3_HBI_System.cRUNNING;
		
		FB_Vacuum_opVacuumOff:= FALSE;
		FB_Vacuum_opVacuumOn:= TRUE;
		FB_Vacuum_fbTimeout(IN:= TRUE, PT:= FB_Vacuum_Timeout, Q=> , ET=> );
		FB_Vacuum_fbSensorDelay(IN:= FB_Vacuum_ipVacuumOn, PT:= FB_Vacuum_SensorDelay, Q=> , ET=> );
		
		IF FB_Vacuum_fbSensorDelay.Q THEN
			FB_Vacuum_M_nVacuumOn_iState:= FB_Vacuum_M_nVacuumOn_iState+1;
			ELSE 
				IF FB_Vacuum_fbTimeout.Q THEN
//					M_nError(nErrorID:= FB_Vacuum_nVacOnAlarmID);
//					FB_Vacuum_sMessage:= CONCAT(CONCAT(UDINT_TO_STRING(FB_Vacuum_nVacOnAlarmID),'>'),
//														CONCAT('>',FB_Vacuum_svacOnAlarmDesc));
					FB_Vacuum_M_nVacuumOn_iState:= 999;
				END_IF
		END_IF
		
	04: // Vacuum done
		M_nVacuumOn:= Tc3_HBI_System.cCOMPLETE;
		
		IF NOT FB_Vacuum_M_nVacuumOn_bExecute THEN
			FB_Vacuum_M_nVacuumOn_iState:= 0;
		END_IF
		
	999: // Error state
		M_nVacuumOn:= Tc3_HBI_System.cABORTED;
		
		FB_Vacuum_opVacuumOff:= FALSE;
		FB_Vacuum_opVacuumOn:= FALSE;
		
		M_nError(nErrorID:= FB_Vacuum_nVacOnAlarmID);
		FB_Vacuum_sMessage:= CONCAT(CONCAT(UDINT_TO_STRING(FB_Vacuum_nVacOnAlarmID),'>'),
											CONCAT('>',FB_Vacuum_svacOnAlarmDesc));
		
		FB_Vacuum_fbTimeout(IN:= FALSE, PT:= T#0S, Q=> , ET=> );
		FB_Vacuum_fbSensorDelay(IN:= FALSE, PT:= T#0S, Q=> , ET=> );
		
		IF NOT FB_Vacuum_M_nVacuumOn_bExecute THEN
			FB_Vacuum_M_nVacuumOn_iState:= 0;
		END_IF
		
	9999: // Parameter error state
		M_nVacuumOn:= Tc3_HBI_System.cPARAMETER_ERROR;
		M_nError(nErrorID:= Tc3_HBI_System.cPARAMETER_ERROR);
		FB_Vacuum_sMessage:= 'Both vacuum on and vacuum off are triggered';
	
ELSE
	FB_Vacuum_M_nVacuumOn_iState:= 00;
	
END_CASE
// =========================================================
END_METHOD

{warning 'add property implementation'}
PROPERTY P_ipVacuumOff : BOOL
GET
P_ipVacuumOff:= FB_Vacuum_ipVacuumOff;
END_GET
SET
FB_Vacuum_ipVacuumOff := P_ipVacuumOff;
END_SET
END_PROPERTY

{warning 'add property implementation'}
PROPERTY P_ipVacuumOn : BOOL
GET
P_ipVacuumOn:= FB_Vacuum_ipVacuumOn;
END_GET
SET
FB_Vacuum_ipVacuumOn := P_ipVacuumOn;
END_SET
END_PROPERTY

{warning 'add property implementation'}
PROPERTY P_nVacOffAlarmID : UDINT
SET
FB_Vacuum_nVacOffAlarmID:= P_nVacOffAlarmID;
END_SET
END_PROPERTY

{warning 'add property implementation'}
PROPERTY P_nVacOnAlarmID : UDINT
SET
FB_Vacuum_nVacOnAlarmID:= P_nVacOnAlarmID;
END_SET
END_PROPERTY

{warning 'add property implementation'}
PROPERTY P_opVacuumOff : BOOL
GET
P_opVacuumOff := FB_Vacuum_opVacuumOff;
END_GET
SET
FB_Vacuum_opVacuumOff:= P_opVacuumOff;
END_SET
END_PROPERTY

{warning 'add property implementation'}
PROPERTY P_opVacuumOn : BOOL
GET
P_opVacuumOn := FB_Vacuum_opVacuumOn;
END_GET
SET
FB_Vacuum_opVacuumOn:= P_opVacuumOn;
END_SET
END_PROPERTY

PROPERTY P_SensorDelay : TIME
SET
FB_Vacuum_SensorDelay:= P_SensorDelay;
END_SET
END_PROPERTY

PROPERTY P_sMessage : STRING
GET
P_sMessage:= FB_Vacuum_sMessage;
END_GET
END_PROPERTY

{warning 'add property implementation'}
PROPERTY P_sVacOffAlarmDesc : STRING
SET
FB_Vacuum_sVacOffAlarmDesc:= P_sVacOffAlarmDesc;
END_SET
END_PROPERTY

{warning 'add property implementation'}
PROPERTY P_sVacOnAlarmDesc : STRING
SET
FB_Vacuum_sVacOnAlarmDesc:= P_sVacOnAlarmDesc;
END_SET
END_PROPERTY

PROPERTY P_Timeout : TIME
SET
FB_Vacuum_Timeout:= P_Timeout;
END_SET
END_PROPERTY

END_FUNCTION_BLOCK

// 06_Purge/ITFs/I_Purge
INTERFACE I_Purge EXTENDS Tc3_HBI_System.I_Basic

METHOD M_nOff : UDINT
VAR_INPUT
END_VAR
END_METHOD

METHOD M_nPurgeOff : UDINT
VAR_INPUT
	bExecute : BOOL;
END_VAR
END_METHOD

METHOD M_nPurgeOn : UDINT
VAR_INPUT
	bExecute: BOOL;
END_VAR
END_METHOD

METHOD M_nSetOutputOff : UDINT
VAR_INPUT
END_VAR
END_METHOD

PROPERTY P_ipPurgeOff : BOOL
GET
END_GET
SET
END_SET
END_PROPERTY

PROPERTY P_ipPurgeOn : BOOL
GET
END_GET
SET
END_SET
END_PROPERTY

PROPERTY P_nPurgeOffAlarmID : UDINT
SET
END_SET
END_PROPERTY

PROPERTY P_nPurgeOnAlarmID : UDINT
SET
END_SET
END_PROPERTY

PROPERTY P_opPurgeOff : BOOL
GET
END_GET
SET
END_SET
END_PROPERTY

PROPERTY P_opPurgeOn : BOOL
GET
END_GET
SET
END_SET
END_PROPERTY

PROPERTY P_SensorDelay : TIME
SET
END_SET
END_PROPERTY

PROPERTY P_sMessage : STRING
GET
END_GET
END_PROPERTY

PROPERTY P_sPurgeOffAlarmDesc : string
SET
END_SET
END_PROPERTY

PROPERTY P_sPurgeOnAlarmDesc : string
SET
END_SET
END_PROPERTY

PROPERTY P_Timeout : TIME
SET
END_SET
END_PROPERTY

END_INTERFACE

// 06_Purge/POUs/FB_Purge
//------------------------------------------------------------------------------------------
//                                                                                        	
//***************************** Beckhoff TwinCAT Examples **********************************
//                                                                                        	
//************************************* WARNING ********************************************
// This program is only an example. If it is used as a control program in any real        	
// application, Beckhoff is not responsible for any malfunction, loss or damage           	
// which could arise by using this program!                                               	
//                                                                                        	
//*************************************  Program Info. *************************************
//                                                                                        	
// PLC program name:       	FB_Purge (FB)                                          	
// Hardware platform:      	TwinCat PTP v3.1.4022				                          	                                  	
//                                                                                        	
// ======================================================================================== 
//         Version       Date                        Remarks                              	
// ======================================================================================== 
//         3.1.1.1      01 March 2018                First release of this example 
//         3.1.1.2      05 March 2018                Next release of this example 
//         3.1.2.1      06 March 2018                Remove purge auto off 
//         3.2.1.1      09 March 2018                Next release of this example   
// ======================================================================================== 
//                                                                                        	
//******************************* Aims OF this PLC PROGRAM *********************************
// 	3.3.1.1 added message for purge alarm                                                                                       	
// 	3.5.3.1 off output once error								 			                                      	
//																	                      	
//                                                                                        	
//----------------------------------------------------------------------------------------- 
FUNCTION_BLOCK FB_Purge EXTENDS FB_Basic IMPLEMENTS I_Purge
VAR 
	FB_Purge_M_nPurgeOff_iState	: INT;
	FB_Purge_M_nPurgeOff_bExecute	: BOOL;
	FB_Purge_M_nPurgeOff_fbExecute_R_TRIG: Tc2_Standard.R_TRIG;
	
	FB_Purge_M_nPurgeOn_iState	: INT;
	FB_Purge_M_nPurgeOn_bExecute	: BOOL;
	FB_Purge_M_nPurgeOn_fbExecute_R_TRIG: Tc2_Standard.R_TRIG;
	
	FB_Purge_M_nReset_iState	: INT;
	FB_Purge_M_nReset_bExecute	: BOOL;
	FB_Purge_M_nReset_fbExecute_R_TRIG: Tc2_Standard.R_TRIG;
	FB_Purge_M_nReset_nStatus	: UDINT;
	
	FB_Purge_ipPurgeOn		: BOOL;
	FB_Purge_ipPurgeOff		: BOOL;
	FB_Purge_opPurgeOn		: BOOL;
	FB_Purge_opPurgeOff		: BOOL;
	FB_Purge_Timeout		: TIME:= T#5S;
	FB_Purge_SensorDelay	: TIME:= T#0MS;
	FB_Purge_sMessage		: STRING(80);
	
	FB_Purge_sPurgeOffAlarmDesc	: STRING(80):='Purge Off Error';
	FB_Purge_sPurgeOnAlarmDesc	: STRING(80):= 'Purge On Error';
	FB_Purge_nPurgeOffAlarmID		: UDINT:= 999;
	FB_Purge_nPurgeOnAlarmID		: UDINT:= 999;
	
	FB_Purge_fbTimeout: Tc2_Standard.TON;
	FB_Purge_fbSensorDelay: Tc2_Standard.TON;
END_VAR

// =========================================================
	
// =========================================================

METHOD M_nOff : UDINT
VAR_INPUT
END_VAR
// =========================================================
M_nPurgeOff(bExecute:= FALSE);
M_nPurgeOn(bExecute:= FALSE);

M_nOff:= Tc3_HBI_System.cCOMPLETE;
// =========================================================
END_METHOD

METHOD M_nPurgeOff : UDINT
VAR_INPUT
	bExecute : BOOL;
END_VAR
// =========================================================
		// Local variables		
FB_Purge_M_nPurgeOff_bExecute:= bExecute;

// =========================================================		
		// Reset
IF _bReset THEN
	IF _bError THEN;
		FB_Purge_sMessage:= '';
		IF FB_Purge_M_nPurgeOff_bExecute THEN
			FB_Purge_M_nPurgeOff_iState:= 01;
			ELSE FB_Purge_M_nPurgeOff_iState:= 00;
		END_IF
	END_IF	
END_IF

// =========================================================
		// Purge off requested
	FB_Purge_M_nPurgeOff_fbExecute_R_TRIG(CLK:= FB_Purge_M_nPurgeOff_bExecute, Q=> );	
	IF FB_Purge_M_nPurgeOff_fbExecute_R_TRIG.Q THEN
		M_nPurgeOn(bExecute:= FALSE);
		FB_Purge_M_nPurgeOff_iState:= 01;
	END_IF

// =========================================================
		// Both purge on and purge off are triggered
	IF FB_Purge_M_nPurgeOff_bExecute AND FB_Purge_M_nPurgeOn_bExecute THEN
		FB_Purge_M_nPurgeOff_iState:= 9999;
	END_IF
		
// =========================================================
		// Purge off state
		
CASE FB_Purge_M_nPurgeOff_iState OF 
	
	00: // Do nothing
		M_nPurgeOff:= Tc3_HBI_System.cIDLE;
		
	01:// Reset timer
		M_nPurgeOff:= Tc3_HBI_System.cRUNNING;
		
		FB_Purge_fbTimeout(IN:= FALSE, PT:= FB_Purge_Timeout, Q=> , ET=> );
		FB_Purge_fbSensorDelay(IN:= FALSE, PT:= FB_Purge_SensorDelay, Q=> , ET=> );
		
		FB_Purge_M_nPurgeOff_iState:= FB_Purge_M_nPurgeOff_iState+1;
		
	02:// Starting
		M_nPurgeOff:= Tc3_HBI_System.cSTARTING;
		
		IF _bReset THEN
			FB_Purge_M_nPurgeOff_iState:= FB_Purge_M_nPurgeOff_iState-1;
			ELSIF FB_Purge_M_nPurgeOff_bExecute THEN
				FB_Purge_M_nPurgeOff_iState:= FB_Purge_M_nPurgeOff_iState+1;
				ELSE FB_Purge_M_nPurgeOff_iState:= 00;
		END_IF
		
	03: // Purge off
		M_nPurgeOff:= Tc3_HBI_System.cRUNNING;
		
		FB_Purge_opPurgeOn:= FALSE;
		FB_Purge_opPurgeOff:= TRUE;
		FB_Purge_fbTimeout(IN:= TRUE, PT:= FB_Purge_Timeout, Q=> , ET=> );
		FB_Purge_fbSensorDelay(IN:= FB_Purge_ipPurgeOff, PT:= FB_Purge_SensorDelay, Q=> , ET=> );
		
		IF FB_Purge_fbSensorDelay.Q THEN
			FB_Purge_M_nPurgeOff_iState:= FB_Purge_M_nPurgeOff_iState+1;
			ELSE 
				IF FB_Purge_fbTimeout.Q THEN
//					M_nError(nErrorID:= FB_Purge_nPurgeOffAlarmID);
//					FB_Purge_sMessage:= CONCAT(CONCAT(UDINT_TO_STRING(FB_Purge_nPurgeOffAlarmID),'>'),
//														CONCAT('>',FB_Purge_sPurgeOffAlarmDesc));
					FB_Purge_M_nPurgeOff_iState:= 999;
				END_IF
		END_IF
		
	04: // Purge done
		M_nPurgeOff:= Tc3_HBI_System.cCOMPLETE;
	
		IF NOT FB_Purge_M_nPurgeOff_bExecute THEN
			FB_Purge_M_nPurgeOff_iState:= 00;
		END_IF
		
	999: // Error state
		M_nPurgeOff:= Tc3_HBI_System.cABORTED;
		
		FB_Purge_opPurgeOn:= FALSE;
		FB_Purge_opPurgeOff:= FALSE;
		
		M_nError(nErrorID:= FB_Purge_nPurgeOffAlarmID);
		FB_Purge_sMessage:= CONCAT(CONCAT(UDINT_TO_STRING(FB_Purge_nPurgeOffAlarmID),'>'),
										CONCAT('>',FB_Purge_sPurgeOffAlarmDesc));
		
		FB_Purge_fbTimeout(IN:= FALSE, PT:= T#0S, Q=> , ET=> );
		FB_Purge_fbSensorDelay(IN:= FALSE, PT:= T#0S, Q=> , ET=> );
		IF NOT FB_Purge_M_nPurgeOff_bExecute THEN
			FB_Purge_M_nPurgeOff_iState:= 00;
		END_IF
		
	9999: // Parameter error state
		M_nPurgeOff:= Tc3_HBI_System.cPARAMETER_ERROR;
		M_nError(nErrorID:= Tc3_HBI_System.cPARAMETER_ERROR);
		FB_Purge_sMessage:= 'Both purge on and purge off are triggered';
			
ELSE
	FB_Purge_M_nPurgeOff_iState:= 00;
	
END_CASE
// =========================================================
END_METHOD

METHOD M_nPurgeOn : UDINT
VAR_INPUT
	bExecute: BOOL;
END_VAR
// =========================================================
		// Local variables		
FB_Purge_M_nPurgeOn_bExecute:= bExecute;

// =========================================================		
		// Reset
IF _bReset THEN
	IF _bError THEN;
		FB_Purge_sMessage:= '';
		IF FB_Purge_M_nPurgeOn_bExecute THEN
			FB_Purge_M_nPurgeOn_iState:= 01;
			ELSE FB_Purge_M_nPurgeOn_iState:= 00;
		END_IF
	END_IF	
END_IF

// =========================================================
	// Purge on requested
	FB_Purge_M_nPurgeOn_fbExecute_R_TRIG(CLK:= FB_Purge_M_nPurgeOn_bExecute, Q=> );
	
	IF FB_Purge_M_nPurgeOn_fbExecute_R_TRIG.Q THEN
		M_nPurgeOff(bExecute:= FALSE);
		FB_Purge_M_nPurgeOn_iState:= 01;
	END_IF

// =========================================================
	// Both purge on and purge off are triggered
	IF FB_Purge_M_nPurgeOff_bExecute AND FB_Purge_M_nPurgeOn_bExecute THEN
		FB_Purge_M_nPurgeOn_iState:= 9999;
	END_IF
		
// =========================================================
		// Purge on state
		
CASE FB_Purge_M_nPurgeOn_iState OF 
	
	00: // Do nothing
		M_nPurgeOn:= Tc3_HBI_System.cIDLE;
		
	01:// Reset timer
		M_nPurgeOn:= Tc3_HBI_System.cRUNNING;
		
		FB_Purge_fbTimeout(IN:= FALSE, PT:= FB_Purge_Timeout, Q=> , ET=> );
		FB_Purge_fbSensorDelay(IN:= FALSE, PT:= FB_Purge_SensorDelay, Q=> , ET=> );
		
		FB_Purge_M_nPurgeOn_iState:= FB_Purge_M_nPurgeOn_iState+1;
		
	02:// Starting
		M_nPurgeOn:= Tc3_HBI_System.cSTARTING;
		
		IF _bReset THEN
			FB_Purge_M_nPurgeOn_iState:= FB_Purge_M_nPurgeOn_iState-1;
			ELSIF FB_Purge_M_nPurgeOn_bExecute THEN
				FB_Purge_M_nPurgeOn_iState:= FB_Purge_M_nPurgeOn_iState+1;
				ELSE FB_Purge_M_nPurgeOn_iState:= 00;
		END_IF
		
	03: // Purge on
		M_nPurgeOn:= Tc3_HBI_System.cRUNNING;
		
		FB_Purge_opPurgeOff:= FALSE;
		FB_Purge_opPurgeOn:= TRUE;
		FB_Purge_fbTimeout(IN:= TRUE, PT:= FB_Purge_Timeout, Q=> , ET=> );
		FB_Purge_fbSensorDelay(IN:= FB_Purge_ipPurgeOn, PT:= FB_Purge_SensorDelay, Q=> , ET=> );
		
		IF FB_Purge_fbSensorDelay.Q THEN
			FB_Purge_M_nPurgeOn_iState:= FB_Purge_M_nPurgeOn_iState+1;
			ELSE 
				IF FB_Purge_fbTimeout.Q THEN
//					M_nError(nErrorID:= FB_Purge_nPurgeOnAlarmID);
//					FB_Purge_sMessage:= CONCAT(CONCAT(UDINT_TO_STRING(FB_Purge_nPurgeOnAlarmID),'>'),
//														CONCAT('>',FB_Purge_sPurgeOnAlarmDesc));
					FB_Purge_M_nPurgeOn_iState:= 999;
				END_IF
		END_IF
		
	04: // Purge done
		M_nPurgeOn:= Tc3_HBI_System.cCOMPLETE;
	
		IF NOT FB_Purge_M_nPurgeOn_bExecute THEN
			FB_Purge_M_nPurgeOn_iState:= 00;
		END_IF
		
	999: // Error state
		M_nPurgeOn:= Tc3_HBI_System.cABORTED;
		
		FB_Purge_opPurgeOff:= FALSE;
		FB_Purge_opPurgeOn:= FALSE;
		
		M_nError(nErrorID:= FB_Purge_nPurgeOnAlarmID);
		FB_Purge_sMessage:= CONCAT(CONCAT(UDINT_TO_STRING(FB_Purge_nPurgeOnAlarmID),'>'),
										CONCAT('>',FB_Purge_sPurgeOnAlarmDesc));
		
		FB_Purge_fbTimeout(IN:= FALSE, PT:= T#0S, Q=> , ET=> );
		FB_Purge_fbSensorDelay(IN:= FALSE, PT:= T#0S, Q=> , ET=> );
		IF NOT FB_Purge_M_nPurgeOn_bExecute THEN
			FB_Purge_M_nPurgeOn_iState:= 00;
		END_IF
		
	9999: // Parameter error state
		M_nPurgeOn:= Tc3_HBI_System.cPARAMETER_ERROR;
		M_nError(nErrorID:= Tc3_HBI_System.cPARAMETER_ERROR);
		FB_Purge_sMessage:= 'Both purge on and purge off are triggered';
			
ELSE
	FB_Purge_M_nPurgeOn_iState:= 00;
	
END_CASE
// =========================================================
END_METHOD

//	The result of the method is an unsigned double integer
//	0 = idle 
//	1 = coupled
//	2 = starting
//	3 = running
//	4 = aborted
// 	5 = no hardware connected
//  6 = Spare
//	7 = pointer or index error
//	8 = mapping error
//	9 = parameter error
//	10 = complete
//	Any other number = ErrorID
METHOD PUBLIC M_nReset : UDINT
VAR_INPUT
	bExecute: BOOL;
END_VAR
// =========================================================
	// Local variables
FB_Purge_M_nReset_bExecute:= bExecute;

// =========================================================	
	// Fire
FB_Purge_M_nReset_fbExecute_R_TRIG(CLK:= FB_Purge_M_nReset_bExecute, Q=> );
IF FB_Purge_M_nReset_fbExecute_R_TRIG.Q THEN
	SUPER^.M_nReset(bExecute:= FALSE);
	FB_Purge_M_nReset_iState:= 01;
END_IF

// =========================================================
	// State machine
	
CASE FB_Purge_M_nReset_iState OF
	00: // Init
		;
		
	01:// Starting
		M_nReset:= Tc3_HBI_System.cSTARTING;
		
		FB_Purge_sMessage:= '';
		
		FB_Purge_M_nPurgeOff_bExecute:= FALSE;
		FB_Purge_M_nPurgeOff_fbExecute_R_TRIG(CLK:= FALSE, Q=> );
		FB_Purge_M_nPurgeOff_iState:= 0;
		
		FB_Purge_M_nPurgeOn_bExecute:= FALSE;
		FB_Purge_M_nPurgeOn_fbExecute_R_TRIG(CLK:= FALSE, Q=> );
		FB_Purge_M_nPurgeOn_iState:= 0;
		
		FB_Purge_M_nReset_iState:= FB_Purge_M_nReset_iState+1;
		
	02:// Running
		M_nReset:= Tc3_HBI_System.cRUNNING;
		
		FB_Purge_M_nReset_nStatus:= SUPER^.M_nReset(bExecute:= TRUE);
		
		// Error 
			IF FB_Purge_M_nReset_nStatus > Tc3_HBI_System.cCOMPLETE THEN
				SUPER^.M_nReset(bExecute:= FALSE);		
				FB_Purge_M_nReset_iState:= FB_Purge_M_nReset_iState+1;
			END_IF

		// Done
			IF FB_Purge_M_nReset_nStatus = Tc3_HBI_System.cCOMPLETE THEN
				SUPER^.M_nReset(bExecute:= FALSE);		
				FB_Purge_M_nReset_iState:= FB_Purge_M_nReset_iState+1;
			END_IF
			
	03: // Done
		M_nReset:= Tc3_HBI_System.cCOMPLETE;
		
			IF NOT FB_Purge_M_nReset_bExecute THEN
				SUPER^.M_nReset(bExecute:= FALSE);		
				FB_Purge_M_nReset_iState:= 000;
			END_IF
	ELSE 
		FB_Purge_M_nReset_iState:= 0;
END_CASE
END_METHOD

METHOD PUBLIC M_nSetOutputOff : UDINT
VAR_INPUT
END_VAR
// =========================================================
FB_Purge_opPurgeOff:= FALSE;
FB_Purge_opPurgeOn:= FALSE;

FB_Purge_M_nPurgeOn_iState:= 0;
FB_Purge_M_nPurgeOff_iState:= 0;

M_nSetOutputOff:= Tc3_HBI_System.cCOMPLETE;
// =========================================================
END_METHOD

PROPERTY PUBLIC P_ipPurgeOff : BOOL
GET
P_ipPurgeOff:= FB_Purge_ipPurgeOff;
END_GET
SET
FB_Purge_ipPurgeOff:= P_ipPurgeOff;
END_SET
END_PROPERTY

PROPERTY PUBLIC P_ipPurgeOn : BOOL
GET
P_ipPurgeOn:= FB_Purge_ipPurgeOn;
END_GET
SET
FB_Purge_ipPurgeOn:= P_ipPurgeOn;
END_SET
END_PROPERTY

{warning 'add property implementation'}
PROPERTY P_nPurgeOffAlarmID : UDINT
SET
FB_Purge_nPurgeOffAlarmID:= P_nPurgeOffAlarmID;
END_SET
END_PROPERTY

{warning 'add property implementation'}
PROPERTY P_nPurgeOnAlarmID : UDINT
SET
FB_Purge_nPurgeOffAlarmID:= P_nPurgeOnAlarmID;
END_SET
END_PROPERTY

{warning 'add property implementation'}
PROPERTY P_opPurgeOff : BOOL
GET
P_opPurgeOff:= FB_Purge_opPurgeOff;
END_GET
SET
FB_Purge_opPurgeOff:= P_opPurgeOff;
END_SET
END_PROPERTY

PROPERTY PUBLIC P_opPurgeOn : BOOL
GET
P_opPurgeOn:= FB_Purge_opPurgeOn;
END_GET
SET
FB_Purge_opPurgeOn:= P_opPurgeOn;
END_SET
END_PROPERTY

PROPERTY P_SensorDelay : TIME
SET
FB_Purge_SensorDelay:= P_SensorDelay;
END_SET
END_PROPERTY

PROPERTY P_sMessage : STRING
GET
P_sMessage:= FB_Purge_sMessage;
END_GET
END_PROPERTY

{warning 'add property implementation'}
PROPERTY P_sPurgeOffAlarmDesc : STRING
SET
FB_Purge_sPurgeOffAlarmDesc:= P_sPurgeOffAlarmDesc;
END_SET
END_PROPERTY

{warning 'add property implementation'}
PROPERTY P_sPurgeOnAlarmDesc : STRING
SET
FB_Purge_sPurgeOnAlarmDesc:= P_sPurgeOnAlarmDesc;
END_SET
END_PROPERTY

PROPERTY P_Timeout : TIME
SET
FB_Purge_Timeout:= P_Timeout;
END_SET
END_PROPERTY

END_FUNCTION_BLOCK

// 07_VacuumPurge/ITFs/I_VacuumPurge
INTERFACE I_VacuumPurge EXTENDS I_Purge, I_Vacuum

METHOD M_nNeutral : UDINT
VAR_INPUT
	bExecute: BOOL;
END_VAR
END_METHOD

METHOD M_nPurgeOn : UDINT
VAR_INPUT
	bExecute: BOOL;
END_VAR
END_METHOD

METHOD M_nVacuumOn : UDINT
VAR_INPUT
	bExecute: BOOL;
END_VAR
END_METHOD

END_INTERFACE

// 07_VacuumPurge/POUs/FB_VacuumPurge
FUNCTION_BLOCK PUBLIC FB_VacuumPurge EXTENDS FB_Basic IMPLEMENTS I_VacuumPurge
VAR_INPUT
END_VAR
VAR_OUTPUT
END_VAR
VAR
// Vacuum instance
	FB_VacuumPurge_fbVacuum: FB_Vacuum;
	FB_VacuumPurge_ipVacuum: I_Vacuum:= FB_VacuumPurge_fbVacuum;
	FB_VacuumPurge_stVacuum: ST_Vacuum;
	FB_VacuumPurge_Vacuum_Timeout		: TIME:= T#5S;
	FB_VacuumPurge_Vacuum_SensorDelay	: TIME:= T#0MS;
	FB_VacuumPurge_Vacuum_fbTimeout: Tc2_Standard.TON;
	FB_VacuumPurge_Vacuum_fbSensorDelay: Tc2_Standard.TON;
// Purge instance
	FB_VacuumPurge_fbPurge: FB_Purge;
	FB_VacuumPurge_ipPurge: I_Purge:= FB_VacuumPurge_fbPurge;
	FB_VacuumPurge_stPurge: ST_Purge;
	FB_VacuumPurge_Purge_Timeout		: TIME:= T#5S;
	FB_VacuumPurge_Purge_SensorDelay	: TIME:= T#0MS;
	FB_VacuumPurge_Purge_fbTimeout: Tc2_Standard.TON;
	FB_VacuumPurge_Purge_fbSensorDelay: Tc2_Standard.TON;
// Local variables
	FB_VacuumPurge_M_nNeutral_iState	: INT;
	FB_VacuumPurge_M_nNeutral_bExecute	: BOOL;
	FB_VacuumPurge_M_nNeutral_fbExecute_R_TRIG: Tc2_Standard.R_TRIG;
		
	FB_VacuumPurge_M_nPurgeOn_iState	: INT;
	FB_VacuumPurge_M_nPurgeOn_bExecute	: BOOL;
	FB_VacuumPurge_M_nPurgeOn_fbExecute_R_TRIG: Tc2_Standard.R_TRIG;
	
	FB_VacuumPurge_M_nVacuumOn_iState	: INT;
	FB_VacuumPurge_M_nVacuumOn_bExecute	: BOOL;
	FB_VacuumPurge_M_nVacuumOn_fbExecute_R_TRIG: Tc2_Standard.R_TRIG;
	
	FB_VacuumPurge_M_nReset_iState	: INT;
	FB_VacuumPurge_M_nReset_bExecute	: BOOL;
	FB_VacuumPurge_M_nReset_fbExecute_R_TRIG: Tc2_Standard.R_TRIG;
	FB_VacuumPurge_M_nReset_nStatus: UDINT;
	
	FB_VacuumPurge_sMessage		: STRING(80);
END_VAR

METHOD PUBLIC M_nNeutral : UDINT
VAR_INPUT
	bExecute: BOOL;
END_VAR
// Local variables
FB_VacuumPurge_M_nNeutral_bExecute:= bExecute;

// Fire
FB_VacuumPurge_M_nNeutral_fbExecute_R_TRIG(CLK:= FB_VacuumPurge_M_nNeutral_bExecute, Q=> );
IF FB_VacuumPurge_M_nNeutral_fbExecute_R_TRIG.Q THEN
	FB_VacuumPurge_M_nNeutral_iState:= 2;
END_IF

// Reset
IF _bReset THEN
	IF _bError THEN
		FB_VacuumPurge_sMessage:='';
		IF FB_VacuumPurge_M_nNeutral_bExecute THEN
			FB_VacuumPurge_M_nNeutral_iState:= 1;
			ELSE FB_VacuumPurge_M_nNeutral_iState:= 0;
		END_IF
	END_IF
END_IF

// State machine
CASE FB_VacuumPurge_M_nNeutral_iState OF 
	0:// Init
		M_nNeutral:= Tc3_HBI_System.cIDLE;
		
	1:// Idle
		M_nNeutral:= Tc3_HBI_System.cIDLE;
		
		FB_VacuumPurge_M_nNeutral_iState:= FB_VacuumPurge_M_nNeutral_iState+1;
		
	2:// Starting
		M_nNeutral:= Tc3_HBI_System.cSTARTING;
		
	3:// Running
		M_nNeutral:= Tc3_HBI_System.cRUNNING;
		
		FB_VacuumPurge_fbPurge.M_nSetOutputOff();
		FB_VacuumPurge_fbVacuum.M_nSetOutputOff();
		
	4:// Complete
		M_nNeutral:= Tc3_HBI_System.cCOMPLETE;
		
		IF NOT FB_VacuumPurge_M_nNeutral_bExecute THEN
			FB_VacuumPurge_M_nNeutral_iState:= 0;
		END_IF
		
	999:// Error state
		M_nNeutral:= Tc3_HBI_System.cABORTED;
		
	ELSE 
		FB_VacuumPurge_M_nNeutral_iState:= 0;
END_CASE
END_METHOD

{warning 'add method implementation'}
METHOD M_nOff : UDINT
END_METHOD

{warning 'add method implementation'}
METHOD M_nPurgeOff : UDINT
VAR_INPUT
	bExecute	: BOOL;
END_VAR
END_METHOD

METHOD PUBLIC M_nPurgeOn : UDINT
VAR_INPUT
	bExecute: BOOL;
END_VAR

VAR
	FB_Vacuum_opPurgeOn: BOOL;
END_VAR
// Local variables
FB_VacuumPurge_M_nPurgeOn_bExecute:= bExecute;

// Fire
FB_VacuumPurge_M_nPurgeOn_fbExecute_R_TRIG(CLK:= FB_VacuumPurge_M_nPurgeOn_bExecute, Q=> );
IF FB_VacuumPurge_M_nPurgeOn_fbExecute_R_TRIG.Q THEN
	FB_VacuumPurge_M_nPurgeOn_iState:= 2;
END_IF

// Reset
IF _bReset THEN
	IF _bError THEN
		FB_VacuumPurge_sMessage:='';
		IF FB_VacuumPurge_M_nPurgeOn_bExecute THEN
			FB_VacuumPurge_M_nPurgeOn_iState:= 1;
			ELSE FB_VacuumPurge_M_nPurgeOn_iState:= 0;
		END_IF
	END_IF
END_IF

// State machine
CASE FB_VacuumPurge_M_nPurgeOn_iState OF 
	0:// Init
		M_nPurgeOn:= Tc3_HBI_System.cIDLE;
		
	1:// Idle
		M_nPurgeOn:= Tc3_HBI_System.cIDLE;
		
		FB_VacuumPurge_M_nPurgeOn_iState:= FB_VacuumPurge_M_nPurgeOn_iState+1;
		
	2:// Starting
		M_nPurgeOn:= TC3_HBI_System.cSTARTING;
		
		IF _bReset THEN
			FB_VacuumPurge_M_nPurgeOn_iState:= FB_VacuumPurge_M_nPurgeOn_iState-1;
			ELSIF FB_VacuumPurge_M_nPurgeOn_bExecute THEN
				FB_VacuumPurge_M_nPurgeOn_iState:= FB_VacuumPurge_M_nPurgeOn_iState+1;
				ELSE FB_VacuumPurge_M_nPurgeOn_iState:= 00;
		END_IF	
		
	3:// Running
		M_nPurgeOn:= TC3_HBI_System.cRUNNING;
		
		IF FB_VacuumPurge_fbPurge.M_nPurgeOn(bExecute:= TRUE)=10 AND FB_VacuumPurge_fbVacuum.M_nVacuumOff(bExecute:= TRUE)=10 THEN
			FB_VacuumPurge_fbPurge.M_nPurgeOn(bExecute:= FALSE);
			FB_VacuumPurge_fbVacuum.M_nVacuumOff(bExecute:= FALSE);
			FB_VacuumPurge_M_nPurgeOn_iState:= FB_VacuumPurge_M_nPurgeOn_iState+1;
			ELSIF FB_VacuumPurge_fbPurge.M_nPurgeOn(bExecute:= TRUE)= 999 THEN
				FB_VacuumPurge_fbVacuum.M_nSetOutputOff();
				FB_VacuumPurge_fbPurge.M_nPurgeOn(bExecute:= FALSE);
				FB_VacuumPurge_fbVacuum.M_nVacuumOff(bExecute:= FALSE);
				FB_VacuumPurge_M_nPurgeOn_iState:= 999;
				ELSIF FB_VacuumPurge_fbVacuum.M_nVacuumOff(bExecute:= TRUE)= 999 THEN
					FB_VacuumPurge_fbPurge.M_nSetOutputOff();
					FB_VacuumPurge_fbPurge.M_nPurgeOn(bExecute:= FALSE);
					FB_VacuumPurge_fbVacuum.M_nVacuumOff(bExecute:= FALSE);
					FB_VacuumPurge_M_nPurgeOn_iState:= 999;
		END_IF
		
	4:// Complete
		M_nPurgeOn:= TC3_HBI_System.cCOMPLETE;
		
		IF NOT FB_VacuumPurge_M_nPurgeOn_bExecute THEN
			FB_VacuumPurge_M_nPurgeOn_iState:= 0;
		END_IF
		
	999:// Error state
		M_nPurgeOn:= Tc3_HBI_System.cABORTED;
		
		IF FB_VacuumPurge_fbPurge.P_nErrorID<> 0 THEN
			M_nError(nErrorID:= FB_VacuumPurge_fbPurge.P_nErrorID);
			FB_VacuumPurge_sMessage:= CONCAT(CONCAT(UDINT_TO_STRING(FB_VacuumPurge_fbPurge.P_nErrorID),'>'),
												CONCAT('>',FB_VacuumPurge_fbPurge.P_sMessage));
			ELSIF FB_VacuumPurge_fbVacuum.P_nErrorID<> 0 THEN
				M_nError(nErrorID:= FB_VacuumPurge_fbVacuum.P_nErrorID);
				FB_VacuumPurge_sMessage:= CONCAT(CONCAT(UDINT_TO_STRING(FB_VacuumPurge_fbVacuum.P_nErrorID),'>'),
													CONCAT('>',FB_VacuumPurge_fbVacuum.P_sMessage));
		END_IF	
		
		IF NOT FB_VacuumPurge_M_nPurgeOn_bExecute THEN
			FB_VacuumPurge_M_nPurgeOn_iState:= 0;
		END_IF
		
	ELSE 
		FB_VacuumPurge_M_nPurgeOn_iState:= 0;
END_CASE
END_METHOD

{warning 'add method implementation'}
METHOD M_nSetOutputOff : UDINT
END_METHOD

{warning 'add method implementation'}
METHOD M_nVacuumOff : UDINT
VAR_INPUT
	bExecute	: BOOL;
END_VAR
END_METHOD

METHOD PUBLIC M_nVacuumOn : UDINT
VAR_INPUT
	bExecute: BOOL;
END_VAR
// Local variables
FB_VacuumPurge_M_nVacuumOn_bExecute:= bExecute;

// Fire
FB_VacuumPurge_M_nVacuumOn_fbExecute_R_TRIG(CLK:= FB_VacuumPurge_M_nVacuumOn_bExecute, Q=> );
IF FB_VacuumPurge_M_nVacuumOn_fbExecute_R_TRIG.Q THEN
	FB_VacuumPurge_M_nVacuumOn_iState:= 2;
END_IF

// Reset
IF _bReset THEN
	IF _bError THEN
		FB_VacuumPurge_sMessage:='';
		IF FB_VacuumPurge_M_nVacuumOn_bExecute THEN
			FB_VacuumPurge_M_nVacuumOn_iState:= 1;
			ELSE FB_VacuumPurge_M_nVacuumOn_iState:= 0;
		END_IF
	END_IF
END_IF

// State machine
CASE FB_VacuumPurge_M_nVacuumOn_iState OF 
	0:// Init
		M_nVacuumOn:= Tc3_HBI_System.cIDLE;
		
	1:// Idle
		M_nVacuumOn:= Tc3_HBI_System.cIDLE;
		
		FB_VacuumPurge_M_nVacuumOn_iState:= FB_VacuumPurge_M_nVacuumOn_iState+1;
		
	2:// Starting
		M_nVacuumOn:= TC3_HBI_System.cSTARTING;
		
		IF _bReset THEN
			FB_VacuumPurge_M_nVacuumOn_iState:= FB_VacuumPurge_M_nVacuumOn_iState-1;
			ELSIF FB_VacuumPurge_M_nVacuumOn_bExecute THEN
				FB_VacuumPurge_M_nVacuumOn_iState:= FB_VacuumPurge_M_nVacuumOn_iState+1;
				ELSE FB_VacuumPurge_M_nVacuumOn_iState:= 00;
		END_IF	
		
	3:// Running
		M_nVacuumOn:= TC3_HBI_System.cRUNNING;
		
		IF FB_VacuumPurge_fbVacuum.M_nVacuumOn(bExecute:= TRUE)=10 AND FB_VacuumPurge_fbPurge.M_nPurgeOff(bExecute:= TRUE)=10 THEN
			FB_VacuumPurge_fbVacuum.M_nVacuumOn(bExecute:= FALSE);
			FB_VacuumPurge_fbPurge.M_nPurgeOff(bExecute:= FALSE);
			FB_VacuumPurge_M_nVacuumOn_iState:= FB_VacuumPurge_M_nVacuumOn_iState+1;
			ELSIF FB_VacuumPurge_fbVacuum.M_nVacuumOn(bExecute:= TRUE)= 999 THEN
				FB_VacuumPurge_fbPurge.M_nSetOutputOff();
				FB_VacuumPurge_fbVacuum.M_nVacuumOn(bExecute:= FALSE);
				FB_VacuumPurge_fbPurge.M_nPurgeOff(bExecute:= FALSE);
				FB_VacuumPurge_M_nVacuumOn_iState:= 999;
				ELSIF FB_VacuumPurge_fbVacuum.M_nVacuumOff(bExecute:= TRUE)= 999 THEN
					FB_VacuumPurge_fbVacuum.M_nVacuumOn(bExecute:= TRUE);
					FB_VacuumPurge_fbVacuum.M_nVacuumOn(bExecute:= FALSE);
					FB_VacuumPurge_fbPurge.M_nPurgeOff(bExecute:= FALSE);
					FB_VacuumPurge_M_nVacuumOn_iState:= 999;
		END_IF
		
	4:// Complete
		M_nVacuumOn:= TC3_HBI_System.cCOMPLETE;
		
		IF NOT FB_VacuumPurge_M_nVacuumOn_bExecute THEN
			FB_VacuumPurge_M_nVacuumOn_iState:= 0;
		END_IF
		
	999:// Error state
		M_nVacuumOn:= Tc3_HBI_System.cABORTED;
		
		IF FB_VacuumPurge_fbVacuum.P_nErrorID<> 0 THEN
			M_nError(nErrorID:= FB_VacuumPurge_fbVacuum.P_nErrorID);
			FB_VacuumPurge_sMessage:= CONCAT(CONCAT(UDINT_TO_STRING(FB_VacuumPurge_fbVacuum.P_nErrorID),'>'),
												CONCAT('>',FB_VacuumPurge_fbVacuum.P_sMessage));
			ELSIF FB_VacuumPurge_fbPurge.P_nErrorID<> 0 THEN
				M_nError(nErrorID:= FB_VacuumPurge_fbPurge.P_nErrorID);
				FB_VacuumPurge_sMessage:= CONCAT(CONCAT(UDINT_TO_STRING(FB_VacuumPurge_fbPurge.P_nErrorID),'>'),
													CONCAT('>',FB_VacuumPurge_fbPurge.P_sMessage));
		END_IF	
		
		IF NOT FB_VacuumPurge_M_nVacuumOn_bExecute THEN
			FB_VacuumPurge_M_nVacuumOn_iState:= 0;
		END_IF
		
	ELSE 
		FB_VacuumPurge_M_nVacuumOn_iState:= 0;
END_CASE
END_METHOD

{warning 'add property implementation'}
PROPERTY P_ipPurgeOff : BOOL
GET
P_ipPurgeOff:= FB_VacuumPurge_fbPurge.P_ipPurgeOff;
END_GET
SET
FB_VacuumPurge_fbPurge.P_ipPurgeOff:= P_ipPurgeOff;
END_SET
END_PROPERTY

{warning 'add property implementation'}
PROPERTY P_ipPurgeOn : BOOL
GET
P_ipPurgeOn:= FB_VacuumPurge_fbPurge.P_ipPurgeOn;
END_GET
SET
FB_VacuumPurge_fbPurge.P_ipPurgeOn:= P_ipPurgeOn;
END_SET
END_PROPERTY

{warning 'add property implementation'}
PROPERTY P_ipVacuumOff : BOOL
GET
P_ipVacuumOff:= FB_VacuumPurge_fbVacuum.P_ipVacuumOff;
END_GET
SET
FB_VacuumPurge_fbVacuum.P_ipVacuumOff:= P_ipVacuumOff;
END_SET
END_PROPERTY

{warning 'add property implementation'}
PROPERTY P_ipVacuumOn : BOOL
GET
P_ipVacuumOn:= FB_VacuumPurge_fbVacuum.P_ipVacuumOn;
END_GET
SET
FB_VacuumPurge_fbVacuum.P_ipVacuumOn:= P_ipVacuumOn;
END_SET
END_PROPERTY

{warning 'add property implementation'}
PROPERTY P_nPurgeOffAlarmID : UDINT
SET
FB_VacuumPurge_fbPurge.P_nPurgeOffAlarmID:= P_nPurgeOffAlarmID;
END_SET
END_PROPERTY

{warning 'add property implementation'}
PROPERTY P_nPurgeOnAlarmID : UDINT
SET
FB_VacuumPurge_fbPurge.P_nPurgeOnAlarmID:= P_nPurgeOnAlarmID;
END_SET
END_PROPERTY

{warning 'add property implementation'}
PROPERTY P_nVacOffAlarmID : UDINT
SET
FB_VacuumPurge_fbVacuum.P_nVacOffAlarmID:= P_nVacOffAlarmID;
END_SET
END_PROPERTY

{warning 'add property implementation'}
PROPERTY P_nVacOnAlarmID : UDINT
SET
FB_VacuumPurge_fbVacuum.P_nVacOnAlarmID:= P_nVacOnAlarmID;
END_SET
END_PROPERTY

{warning 'add property implementation'}
PROPERTY P_opPurgeOff : BOOL
GET
P_opPurgeOff:= FB_VacuumPurge_fbPurge.P_opPurgeOff;
END_GET
SET
FB_VacuumPurge_fbPurge.P_opPurgeOff:= P_opPurgeOff;
END_SET
END_PROPERTY

{warning 'add property implementation'}
PROPERTY P_opPurgeOn : BOOL
GET
P_opPurgeOn:= FB_VacuumPurge_fbPurge.P_opPurgeOn;
END_GET
SET
FB_VacuumPurge_fbPurge.P_opPurgeOn:= P_opPurgeOn;
END_SET
END_PROPERTY

{warning 'add property implementation'}
PROPERTY P_opVacuumOff : BOOL
GET
P_opVacuumOff:= FB_VacuumPurge_fbVacuum.P_opVacuumOff;
END_GET
SET
FB_VacuumPurge_fbVacuum.P_opVacuumOff:= P_opVacuumOff;
END_SET
END_PROPERTY

{warning 'add property implementation'}
PROPERTY P_opVacuumOn : BOOL
GET
P_opVacuumOn:= FB_VacuumPurge_fbVacuum.P_opVacuumOn;
END_GET
SET
FB_VacuumPurge_fbVacuum.P_opVacuumOn:= P_opVacuumOn;
END_SET
END_PROPERTY

PROPERTY PUBLIC P_PurgeTimeout : TIME
GET
END_GET
SET
END_SET
END_PROPERTY

{warning 'add property implementation'}
PROPERTY P_SensorDelay : TIME
SET
END_SET
END_PROPERTY

{warning 'add property implementation'}
PROPERTY P_sMessage : STRING
GET
END_GET
END_PROPERTY

{warning 'add property implementation'}
PROPERTY P_sPurgeOffAlarmDesc : STRING
SET
FB_VacuumPurge_fbPurge.P_sPurgeOffAlarmDesc:= P_sPurgeOffAlarmDesc;
END_SET
END_PROPERTY

{warning 'add property implementation'}
PROPERTY P_sPurgeOnAlarmDesc : STRING
SET
FB_VacuumPurge_fbPurge.P_sPurgeOnAlarmDesc:= P_sPurgeOnAlarmDesc;
END_SET
END_PROPERTY

{warning 'add property implementation'}
PROPERTY P_sVacOffAlarmDesc : STRING
SET
FB_VacuumPurge_fbVacuum.P_sVacOffAlarmDesc:= P_sVacOffAlarmDesc;
END_SET
END_PROPERTY

{warning 'add property implementation'}
PROPERTY P_sVacOnAlarmDesc : STRING
SET
FB_VacuumPurge_fbVacuum.P_sVacOnAlarmDesc:= P_sVacOnAlarmDesc;
END_SET
END_PROPERTY

{warning 'add property implementation'}
PROPERTY P_Timeout : TIME
SET
END_SET
END_PROPERTY

PROPERTY PUBLIC P_VacuumTimeout : TIME
GET
END_GET
SET
END_SET
END_PROPERTY

END_FUNCTION_BLOCK
